FUNCTION_BLOCK B_1Event_10States (* Basic FB with empty ECC *)
  (* Standard: 61499-2 *)
  (* Version 1.0, 2023-09-22, AK124910 *)
  PACKAGE servSeq;
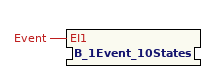
  EVENT_INPUT
    EI1;
  END_EVENT
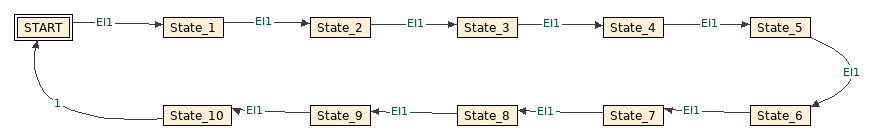
  EC_STATES
    START; (* Initial State *)
    State_1;
    State_2;
    State_3;
    State_4;
    State_5;
    State_6;
    State_7;
    State_8;
    State_9;
    State_10;
  END_STATES
  EC_TRANSITIONS
    START TO State_1 := EI1;
    State_1 TO State_2 := EI1;
    State_2 TO State_3 := EI1;
    State_3 TO State_4 := EI1;
    State_4 TO State_5 := EI1;
    State_5 TO State_6 := EI1;
    State_6 TO State_7 := EI1;
    State_7 TO State_8 := EI1;
    State_8 TO State_9 := EI1;
    State_9 TO State_10 := EI1;
    State_10 TO START := 1;
  END_TRANSITIONS
  (* Service external/internal_interface: Basic FB with empty ECC *)
END_FUNCTION_BLOCK
